PROGRAM MAIN
VAR
END_VAR

END_PROGRAM

(* stored: Version 1.1.0.1
   POU MAIN: Id {87d6bba0-cac0-4c5b-b8ef-b01bdb9ad7f6} *)
